(* IEC 61131-3 sources: InfiniteStateMachine/extracted_st/library_information/getlibversionnumber, 1 file *)

(* ---- GetLibVersionNumber.st ---- *)
(* --- Interface --- *)
// This function has been automatically generated from the project information.
FUNCTION GetLibVersionNumber : DWORD
VAR_INPUT

END_VAR
(* --- Implementation --- *)
GetLibVersionNumber := 65793;
